// TIA Portal V18 export
// export: Created 2025-12-01T12:38:34.7505824Z, ExportSetting None, DisplayName Totally Integrated Automation Portal, DisplayVersion V18 Update 5, DisplayName TIA Portal Openness, DisplayVersion V18 Update 5, DisplayName TIA Portal Teamcenter Gateway, DisplayVersion V18, DisplayName TIA Portal Version Control Interface, DisplayVersion V18, DisplayName STEP 7 Professional, DisplayVersion V18 Update 5, DisplayName STEP 7 Safety, DisplayVersion V18, DisplayName WinCC Professional, DisplayVersion V18 Update 5
DATA_BLOCK "ST10_Stopper_FB_DB"   // DB1160
// stored: AutoNumber false, InstanceOfName ST10_Stopper_FB, InstanceOfType FB
"ST10_Stopper_FB"
   // VAR
   //    FB_Stopper_Instance { S7_SetPoint := 'True'} : Array[1..3] of "FB_Stopper";
   // END_VAR
BEGIN
END_DATA_BLOCK
